// TIA Portal V17 export
FUNCTION "MotorControl" : Void   // FC, LAD
{ S7_Optimized_Access := 'TRUE' }
VERSION : 0.1
// stored: AutoNumber true, IsIECCheckEnabled false, SetENOAutomatically false
BEGIN

REGION Network 1
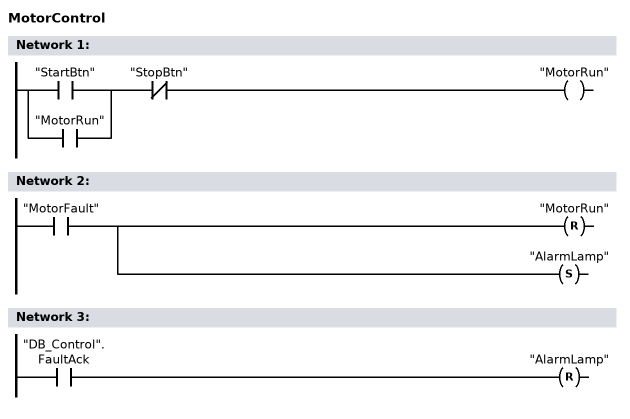
   RUNG wire#powerrail
      Contact( "StartBtn" )
      wire#w1
      I_Contact( "StopBtn" )
      Coil( "MotorRun" )
   END_RUNG
   RUNG wire#powerrail
      Contact( "MotorRun" )
   END_RUNG wire#w1
   // the same network as SCL:
   "MotorRun" := ("StartBtn" OR "MotorRun") AND NOT "StopBtn";
END_REGION

REGION Network 2
   RUNG wire#powerrail
      Contact( "MotorFault" )
      wire#w1
      R_Coil( "MotorRun" )
   END_RUNG
   RUNG wire#w1
      S_Coil( "AlarmLamp" )
   END_RUNG
   // the same network as SCL:
   IF "MotorFault" THEN
       "MotorRun" := FALSE;
       "AlarmLamp" := TRUE;
   END_IF;
END_REGION

REGION Network 3
   RUNG wire#powerrail
      Contact( "DB_Control".FaultAck )
      R_Coil( "AlarmLamp" )
   END_RUNG
   // the same network as SCL:
   IF "DB_Control".FaultAck THEN "AlarmLamp" := FALSE; END_IF;
END_REGION
END_FUNCTION
